// TIA Portal V21 export
DATA_BLOCK "VistaManuali"   // DB31
{ S7_Optimized_Access := 'TRUE' }
// stored: MemoryReserve 100
   VAR RETAIN
      VistaManuale : Array[0.."K_NumVistaManuale"] of Struct
         K_Tipo : Int;
         K_NumeroUtenza : Int;
      END_STRUCT;
   END_VAR
BEGIN
   VistaManuale[0].K_Tipo := 0;
   VistaManuale[0].K_NumeroUtenza := 0;
END_DATA_BLOCK
